FUNCTION TryConvert_DINT_TO_ULINT : BOOL
VAR_INPUT
	in : DINT;
	out : REFERENCE TO ULINT;
END_VAR

IF in < DatatypeLimits.MIN_VALUE_OF_DINT_WHICH_CAN_BE_HELD_IN_A_ULINT THEN
	RETURN;
END_IF

out := DINT_TO_ULINT(in);
TryConvert_DINT_TO_ULINT := TRUE;

END_FUNCTION

(* stored: Version 1.1.0.1, ProductVersion 3.1.4024.12
   POU TryConvert_DINT_TO_ULINT: Id {a42aa242-cce2-42af-b3d7-33e77e2fdf76}, SpecialFunc None *)
